Staubli VAL3: D_ABZ_00.dtx

public aio aiEncCurrentPos = {link=e00CurrPos}
aio aiEncLatchedPos = {link=e00LatchPos}
aio aoEncResolution = {link=e00Counts}
aio aoPresetPos = {link=e00PrstPos}
public bool bLatchEnabled = true
bool bLatchLevel = true
bool bMemoLatchState
bool bPartLatched
bool bReset
dio diEncHwErr = {link=e00HwErr}
dio diEncLatched = {link=e00Latch}
dio diEncOvsErr = {link=e00OvsErr}
dio diLatchSignal = {link=e00LatchSig}
dio doEnableLatch = {link=e00EnLatch}
dio doEnablePreset = {link=e00EnPrst}
dio doLatchEdgFall = {link=e00LatchEdgFall}
dio doResetErr = {link=e00RstErr}
num nEncLatchedVal
num nEncResolution = 2000
num nEncValue = 612
public num nLatchPeriod = 1
public num nMAXCOUNT = 96636764.16
public num nMINCOUNT = -96636764.16
num nPresetPos
string sEncNum = "ENC0"
string sTASK = "encoder0"
